//Verdichter zählen
	Count(
	x_Ein_1:= x_Aus1, 
	x_Ein_2:= x_Aus2, 
	x_Ein_3:= x_Aus3, 
	x_Ein_4:= x_Aus4,
	x_Ein_5:= x_Aus5,
	x_Ein_6:= x_Aus6,
	x_Ein_7:= x_Aus7,
	x_Ein_8:= x_Aus8,
	i_Aus=> i_Count);
//Betriebsstunden vergleichen
	//Vergleich zu Verdichter 1
	x_1_2(t_Ein1:=t_Betriebsstunden1, t_Ein2:= t_Betriebsstunden2);
	x_1_3(t_Ein1:=t_Betriebsstunden1, t_Ein2:= t_Betriebsstunden3);
	x_1_4(t_Ein1:=t_Betriebsstunden1, t_Ein2:= t_Betriebsstunden4);
	x_1_5(t_Ein1:=t_Betriebsstunden1, t_Ein2:= t_Betriebsstunden5);
	x_1_6(t_Ein1:=t_Betriebsstunden1, t_Ein2:= t_Betriebsstunden6);
	x_1_7(t_Ein1:=t_Betriebsstunden1, t_Ein2:= t_Betriebsstunden7);
	x_1_8(t_Ein1:=t_Betriebsstunden1, t_Ein2:= t_Betriebsstunden8);
	//Vergleich zu Verdichter 2
	x_2_1(t_Ein1:=t_Betriebsstunden2, t_Ein2:= t_Betriebsstunden1);
	x_2_3(t_Ein1:=t_Betriebsstunden2, t_Ein2:= t_Betriebsstunden3);
	x_2_4(t_Ein1:=t_Betriebsstunden2, t_Ein2:= t_Betriebsstunden4);
	x_2_5(t_Ein1:=t_Betriebsstunden2, t_Ein2:= t_Betriebsstunden5);
	x_2_6(t_Ein1:=t_Betriebsstunden2, t_Ein2:= t_Betriebsstunden6);
	x_2_7(t_Ein1:=t_Betriebsstunden2, t_Ein2:= t_Betriebsstunden7);
	x_2_8(t_Ein1:=t_Betriebsstunden2, t_Ein2:= t_Betriebsstunden8);
	//Vergleich zu Verdichter 3
	x_3_1(t_Ein1:=t_Betriebsstunden3, t_Ein2:= t_Betriebsstunden1);
	x_3_2(t_Ein1:=t_Betriebsstunden3, t_Ein2:= t_Betriebsstunden2);
	x_3_4(t_Ein1:=t_Betriebsstunden3, t_Ein2:= t_Betriebsstunden4);
	x_3_5(t_Ein1:=t_Betriebsstunden3, t_Ein2:= t_Betriebsstunden5);
	x_3_6(t_Ein1:=t_Betriebsstunden3, t_Ein2:= t_Betriebsstunden6);
	x_3_7(t_Ein1:=t_Betriebsstunden3, t_Ein2:= t_Betriebsstunden7);
	x_3_8(t_Ein1:=t_Betriebsstunden3, t_Ein2:= t_Betriebsstunden8);
	//Vergleich zu Verdichter 4
	x_4_1(t_Ein1:=t_Betriebsstunden4, t_Ein2:= t_Betriebsstunden1);
	x_4_2(t_Ein1:=t_Betriebsstunden4, t_Ein2:= t_Betriebsstunden2);
	x_4_3(t_Ein1:=t_Betriebsstunden4, t_Ein2:= t_Betriebsstunden3);
	x_4_5(t_Ein1:=t_Betriebsstunden4, t_Ein2:= t_Betriebsstunden5);
	x_4_6(t_Ein1:=t_Betriebsstunden4, t_Ein2:= t_Betriebsstunden6);
	x_4_7(t_Ein1:=t_Betriebsstunden4, t_Ein2:= t_Betriebsstunden7);
	x_4_8(t_Ein1:=t_Betriebsstunden4, t_Ein2:= t_Betriebsstunden8);
	//Vergleich zu Verdichter 5
	x_5_1(t_Ein1:=t_Betriebsstunden5, t_Ein2:= t_Betriebsstunden1);
	x_5_2(t_Ein1:=t_Betriebsstunden5, t_Ein2:= t_Betriebsstunden2);
	x_5_3(t_Ein1:=t_Betriebsstunden5, t_Ein2:= t_Betriebsstunden3);
	x_5_4(t_Ein1:=t_Betriebsstunden5, t_Ein2:= t_Betriebsstunden4);
	x_5_6(t_Ein1:=t_Betriebsstunden5, t_Ein2:= t_Betriebsstunden6);
	x_5_7(t_Ein1:=t_Betriebsstunden5, t_Ein2:= t_Betriebsstunden7);
	x_5_8(t_Ein1:=t_Betriebsstunden5, t_Ein2:= t_Betriebsstunden8);
	//Vergleich zu Verdichter 6
	x_6_1(t_Ein1:=t_Betriebsstunden6, t_Ein2:= t_Betriebsstunden1);
	x_6_2(t_Ein1:=t_Betriebsstunden6, t_Ein2:= t_Betriebsstunden2);
	x_6_3(t_Ein1:=t_Betriebsstunden6, t_Ein2:= t_Betriebsstunden3);
	x_6_4(t_Ein1:=t_Betriebsstunden6, t_Ein2:= t_Betriebsstunden4);
	x_6_5(t_Ein1:=t_Betriebsstunden6, t_Ein2:= t_Betriebsstunden5);
	x_6_7(t_Ein1:=t_Betriebsstunden6, t_Ein2:= t_Betriebsstunden7);
	x_6_8(t_Ein1:=t_Betriebsstunden6, t_Ein2:= t_Betriebsstunden8);
	//Vergleich zu Verdichter 7
	x_7_1(t_Ein1:=t_Betriebsstunden7, t_Ein2:= t_Betriebsstunden1);
	x_7_2(t_Ein1:=t_Betriebsstunden7, t_Ein2:= t_Betriebsstunden2);
	x_7_3(t_Ein1:=t_Betriebsstunden7, t_Ein2:= t_Betriebsstunden3);
	x_7_4(t_Ein1:=t_Betriebsstunden7, t_Ein2:= t_Betriebsstunden4);
	x_7_5(t_Ein1:=t_Betriebsstunden7, t_Ein2:= t_Betriebsstunden5);
	x_7_6(t_Ein1:=t_Betriebsstunden7, t_Ein2:= t_Betriebsstunden6);
	x_7_8(t_Ein1:=t_Betriebsstunden7, t_Ein2:= t_Betriebsstunden8);
	//Vergleich zu Verdichter 8
	x_8_1(t_Ein1:=t_Betriebsstunden8, t_Ein2:= t_Betriebsstunden1);
	x_8_2(t_Ein1:=t_Betriebsstunden8, t_Ein2:= t_Betriebsstunden2);
	x_8_3(t_Ein1:=t_Betriebsstunden8, t_Ein2:= t_Betriebsstunden3);
	x_8_4(t_Ein1:=t_Betriebsstunden8, t_Ein2:= t_Betriebsstunden4);
	x_8_5(t_Ein1:=t_Betriebsstunden8, t_Ein2:= t_Betriebsstunden5);
	x_8_6(t_Ein1:=t_Betriebsstunden8, t_Ein2:= t_Betriebsstunden6);
	x_8_7(t_Ein1:=t_Betriebsstunden8, t_Ein2:= t_Betriebsstunden7);
	
//Verdichterumschaltung für einen Zyklus einen Verdichter mehr anfordern Umschaltung verläuft also quasi nahtlos
	IF x_Wechsel AND NOT x_Speicher THEN
		i_Stufen:= i_Stufen+1;
	END_IF
	x_Speicher:=x_Wechsel;
	
//Einschalten
	//Einschalten Verdichter 1
		IF x_En1 AND i_Stufen > i_Count AND NOT x_Aus1 AND
			(x_1_2.x_Aus AND x_En2 OR x_Aus2 OR NOT x_En2) AND
			(x_1_3.x_Aus AND x_En3 OR x_Aus3 OR NOT x_En3) AND
			(x_1_4.x_Aus AND x_En4 OR x_Aus4 OR NOT x_En4) AND
			(x_1_5.x_Aus AND x_En5 OR x_Aus5 OR NOT x_En5) AND
			(x_1_6.x_Aus AND x_En6 OR x_Aus6 OR NOT x_En6) AND
			(x_1_7.x_Aus AND x_En7 OR x_Aus7 OR NOT x_En7) AND
			(x_1_8.x_Aus AND x_En8 OR x_Aus8 OR NOT x_En8) THEN
			x_Aus1:=TRUE;
			t_Ein1:=Globale_Uhr.systemDateAndTime;
			i_Count:=i_Count+1;
		END_IF
	
	//Einschalten Verdichter 2
		IF x_En2 AND i_Stufen > i_Count AND NOT x_Aus2 AND
			(x_2_1.x_Aus AND x_En1 OR x_Aus1 OR NOT x_En1) AND
			(x_2_3.x_Aus AND x_En3 OR x_Aus3 OR NOT x_En3) AND
			(x_2_4.x_Aus AND x_En4 OR x_Aus4 OR NOT x_En4) AND
			(x_2_5.x_Aus AND x_En5 OR x_Aus5 OR NOT x_En5) AND
			(x_2_6.x_Aus AND x_En6 OR x_Aus6 OR NOT x_En6) AND
			(x_2_7.x_Aus AND x_En7 OR x_Aus7 OR NOT x_En7) AND
			(x_2_8.x_Aus AND x_En8 OR x_Aus8 OR NOT x_En8) THEN
			x_Aus2:=TRUE;
			t_Ein2:=Globale_Uhr.systemDateAndTime;
			i_Count:=i_Count+1;
		END_IF	
	
	//Einschalten Verdichter 3
		IF x_En3 AND i_Stufen > i_Count AND NOT x_Aus3 AND
			(x_3_1.x_Aus AND x_En1 OR x_Aus1 OR NOT x_En1) AND
			(x_3_2.x_Aus AND x_En2 OR x_Aus2 OR NOT x_En2) AND
			(x_3_4.x_Aus AND x_En4 OR x_Aus4 OR NOT x_En4) AND
			(x_3_5.x_Aus AND x_En5 OR x_Aus5 OR NOT x_En5) AND
			(x_3_6.x_Aus AND x_En6 OR x_Aus6 OR NOT x_En6) AND
			(x_3_7.x_Aus AND x_En7 OR x_Aus7 OR NOT x_En7) AND
			(x_3_8.x_Aus AND x_En8 OR x_Aus8 OR NOT x_En8) THEN
			x_Aus3:=TRUE;
			t_Ein3:=Globale_Uhr.systemDateAndTime;
			i_Count:=i_Count+1;
		END_IF	
	
	//Einschalten Verdichter 4
		IF x_En4 AND i_Stufen > i_Count AND NOT x_Aus4 AND 
			(x_4_1.x_Aus AND x_En1 OR x_Aus1 OR NOT x_En1) AND
			(x_4_2.x_Aus AND x_En2 OR x_Aus2 OR NOT x_En2) AND
			(x_4_3.x_Aus AND x_En3 OR x_Aus3 OR NOT x_En3) AND
			(x_4_5.x_Aus AND x_En5 OR x_Aus5 OR NOT x_En5) AND
			(x_4_6.x_Aus AND x_En6 OR x_Aus6 OR NOT x_En6) AND
			(x_4_7.x_Aus AND x_En7 OR x_Aus7 OR NOT x_En7) AND
			(x_4_8.x_Aus AND x_En8 OR x_Aus8 OR NOT x_En8) THEN
			x_Aus4:=TRUE;
			t_Ein4:=Globale_Uhr.systemDateAndTime;
			i_Count:=i_Count+1;
		END_IF	
	//Einschalten Verdichter 5
		IF x_En5 AND i_Stufen > i_Count AND NOT x_Aus5 AND
			(x_5_1.x_Aus AND x_En1 OR x_Aus1 OR NOT x_En1) AND
			(x_5_2.x_Aus AND x_En2 OR x_Aus2 OR NOT x_En2) AND
			(x_5_3.x_Aus AND x_En3 OR x_Aus3 OR NOT x_En3) AND
			(x_5_4.x_Aus AND x_En4 OR x_Aus4 OR NOT x_En4) AND
			(x_5_6.x_Aus AND x_En6 OR x_Aus6 OR NOT x_En6) AND
			(x_5_7.x_Aus AND x_En7 OR x_Aus7 OR NOT x_En7) AND
			(x_5_8.x_Aus AND x_En8 OR x_Aus8 OR NOT x_En8) THEN
			x_Aus5:=TRUE;
			t_Ein5:=Globale_Uhr.systemDateAndTime;
			i_Count:=i_Count+1;
		END_IF
	
	//Einschalten Verdichter 6
		IF x_En6 AND i_Stufen > i_Count AND NOT x_Aus6 AND
			(x_6_1.x_Aus AND x_En1 OR x_Aus1 OR NOT x_En1) AND
			(x_6_2.x_Aus AND x_En2 OR x_Aus2 OR NOT x_En2) AND
			(x_6_3.x_Aus AND x_En3 OR x_Aus3 OR NOT x_En3) AND
			(x_6_4.x_Aus AND x_En4 OR x_Aus4 OR NOT x_En4) AND
			(x_6_5.x_Aus AND x_En5 OR x_Aus5 OR NOT x_En5) AND
			(x_6_7.x_Aus AND x_En7 OR x_Aus7 OR NOT x_En7) AND
			(x_6_8.x_Aus AND x_En8 OR x_Aus8 OR NOT x_En8) THEN
			x_Aus6:=TRUE;
			t_Ein6:=Globale_Uhr.systemDateAndTime;
			i_Count:=i_Count+1;
		END_IF	
	
	//Einschalten Verdichter 7
		IF x_En7 AND i_Stufen > i_Count AND NOT x_Aus7 AND
			(x_7_1.x_Aus AND x_En1 OR x_Aus1 OR NOT x_En1) AND
			(x_7_2.x_Aus AND x_En2 OR x_Aus2 OR NOT x_En2) AND
			(x_7_3.x_Aus AND x_En3 OR x_Aus3 OR NOT x_En3) AND
			(x_7_4.x_Aus AND x_En4 OR x_Aus4 OR NOT x_En4) AND
			(x_7_5.x_Aus AND x_En5 OR x_Aus5 OR NOT x_En5) AND
			(x_7_6.x_Aus AND x_En6 OR x_Aus6 OR NOT x_En6) AND
			(x_7_8.x_Aus AND x_En8 OR x_Aus8 OR NOT x_En8) THEN
			x_Aus7:=TRUE;
			t_Ein7:=Globale_Uhr.systemDateAndTime;
			i_Count:=i_Count+1;
		END_IF	
	
	//Einschalten Verdichter 8
		IF x_En8 AND i_Stufen > i_Count AND NOT x_Aus8 AND
			(x_8_1.x_Aus AND x_En1 OR x_Aus1 OR NOT x_En1) AND
			(x_8_2.x_Aus AND x_En2 OR x_Aus2 OR NOT x_En2) AND
			(x_8_3.x_Aus AND x_En3 OR x_Aus3 OR NOT x_En3) AND
			(x_8_4.x_Aus AND x_En4 OR x_Aus4 OR NOT x_En4) AND
			(x_8_5.x_Aus AND x_En5 OR x_Aus5 OR NOT x_En5) AND
			(x_8_6.x_Aus AND x_En6 OR x_Aus6 OR NOT x_En6) AND
			(x_8_7.x_Aus AND x_En7 OR x_Aus7 OR NOT x_En7) THEN
			x_Aus8:=TRUE;
			t_Ein8:=Globale_Uhr.systemDateAndTime;
			i_Count:=i_Count+1;
		END_IF	
	
//Ausschalten
	//Ausschalten Verdichter 1
		IF NOT x_En1 AND x_Aus1 OR (i_Stufen < i_Count AND x_Aus1 AND
			//(t_Ein1 <= t_Ein1 OR NOT x_Aus1) AND
			(t_Ein1 <= t_Ein2 OR NOT x_Aus2) AND
			(t_Ein1 <= t_Ein3 OR NOT x_Aus3) AND
			(t_Ein1 <= t_Ein4 OR NOT x_Aus4) AND
			(t_Ein1 <= t_Ein5 OR NOT x_Aus5) AND
			(t_Ein1 <= t_Ein6 OR NOT x_Aus6) AND
			(t_Ein1 <= t_Ein7 OR NOT x_Aus7) AND
			(t_Ein1 <= t_Ein8 OR NOT x_Aus8)) THEN
			x_Aus1:=FALSE;
			i_Count:= i_Count-1;
		END_IF	
		
	//Ausschalten Verdichter 2
		IF NOT x_En2 AND x_Aus2 OR (i_Stufen < i_Count AND x_Aus2 AND
			(t_Ein2 <= t_Ein1 OR NOT x_Aus1) AND
			//(t_Ein2 <= t_Ein2 OR NOT x_Aus2) AND
			(t_Ein2 <= t_Ein3 OR NOT x_Aus3) AND
			(t_Ein2 <= t_Ein4 OR NOT x_Aus4) AND
			(t_Ein2 <= t_Ein5 OR NOT x_Aus5) AND
			(t_Ein2 <= t_Ein6 OR NOT x_Aus6) AND
			(t_Ein2 <= t_Ein7 OR NOT x_Aus7) AND
			(t_Ein2 <= t_Ein8 OR NOT x_Aus8)) THEN
			x_Aus2:=FALSE;
			i_Count:= i_Count-1;
		END_IF	
		
	//Ausschalten Verdichter 3
		IF NOT x_En3 AND x_Aus3 OR (i_Stufen < i_Count AND x_Aus3 AND
			(t_Ein3 <= t_Ein1 OR NOT x_Aus1) AND
			(t_Ein3 <= t_Ein2 OR NOT x_Aus2) AND
			//(t_Ein3 <= t_Ein3 OR NOT x_Aus3) AND
			(t_Ein3 <= t_Ein4 OR NOT x_Aus4) AND
			(t_Ein3 <= t_Ein5 OR NOT x_Aus5) AND
			(t_Ein3 <= t_Ein6 OR NOT x_Aus6) AND
			(t_Ein3 <= t_Ein7 OR NOT x_Aus7) AND
			(t_Ein3 <= t_Ein8 OR NOT x_Aus8)) THEN
			x_Aus3:=FALSE;
			i_Count:= i_Count-1;
		END_IF	
		
	//Ausschalten Verdichter 4
		IF NOT x_En4 AND x_Aus4 OR (i_Stufen < i_Count AND x_Aus4 AND
			(t_Ein4 <= t_Ein1 OR NOT x_Aus1) AND
			(t_Ein4 <= t_Ein2 OR NOT x_Aus2) AND
			(t_Ein4 <= t_Ein3 OR NOT x_Aus3) AND
			//(t_Ein4 <= t_Ein4 OR NOT x_Aus4) AND
			(t_Ein4 <= t_Ein5 OR NOT x_Aus5) AND
			(t_Ein4 <= t_Ein6 OR NOT x_Aus6) AND
			(t_Ein4 <= t_Ein7 OR NOT x_Aus7) AND
			(t_Ein4 <= t_Ein8 OR NOT x_Aus8)) THEN
			x_Aus4:=FALSE;
			i_Count:= i_Count-1;
		END_IF	
		
	//Ausschalten Verdichter 5
		IF NOT x_En5 AND x_Aus5 OR (i_Stufen < i_Count AND x_Aus5 AND
			(t_Ein5 <= t_Ein1 OR NOT x_Aus1) AND
			(t_Ein5 <= t_Ein2 OR NOT x_Aus2) AND
			(t_Ein5 <= t_Ein3 OR NOT x_Aus3) AND
			(t_Ein5 <= t_Ein4 OR NOT x_Aus4) AND
			//(t_Ein5 <= t_Ein5 OR NOT x_Aus5) AND
			(t_Ein5 <= t_Ein6 OR NOT x_Aus6) AND
			(t_Ein5 <= t_Ein7 OR NOT x_Aus7) AND
			(t_Ein5 <= t_Ein8 OR NOT x_Aus8)) THEN
			x_Aus5:=FALSE;
			i_Count:= i_Count-1;
		END_IF		
		
	//Ausschalten Verdichter 6
		IF NOT x_En6 AND x_Aus6 OR (i_Stufen < i_Count AND x_Aus6 AND
			(t_Ein6 <= t_Ein1 OR NOT x_Aus1) AND
			(t_Ein6 <= t_Ein2 OR NOT x_Aus2) AND
			(t_Ein6 <= t_Ein3 OR NOT x_Aus3) AND
			(t_Ein6 <= t_Ein4 OR NOT x_Aus4) AND
			(t_Ein6 <= t_Ein5 OR NOT x_Aus5) AND
			//(t_Ein6 <= t_Ein6 OR NOT x_Aus6) AND
			(t_Ein6 <= t_Ein7 OR NOT x_Aus7) AND
			(t_Ein6 <= t_Ein8 OR NOT x_Aus8)) THEN
			x_Aus6:=FALSE;
			i_Count:= i_Count-1;
		END_IF	
		
	//Ausschalten Verdichter 7
		IF NOT x_En7 AND x_Aus7 OR (i_Stufen < i_Count AND x_Aus7 AND
			(t_Ein7 <= t_Ein1 OR NOT x_Aus1) AND
			(t_Ein7 <= t_Ein2 OR NOT x_Aus2) AND
			(t_Ein7 <= t_Ein3 OR NOT x_Aus3) AND
			(t_Ein7 <= t_Ein4 OR NOT x_Aus4) AND
			(t_Ein7 <= t_Ein5 OR NOT x_Aus5) AND
			(t_Ein7 <= t_Ein6 OR NOT x_Aus6) AND
			//(t_Ein7 <= t_Ein7 OR NOT x_Aus7) AND
			(t_Ein7 <= t_Ein8 OR NOT x_Aus8)) THEN
			x_Aus7:=FALSE;
			i_Count:= i_Count-1;
		END_IF	
		
	//Ausschalten Verdichter 8
		IF NOT x_En8 AND x_Aus8 OR (i_Stufen < i_Count AND x_Aus8 AND
			(t_Ein8 <= t_Ein1 OR NOT x_Aus1) AND
			(t_Ein8 <= t_Ein2 OR NOT x_Aus2) AND
			(t_Ein8 <= t_Ein3 OR NOT x_Aus3) AND
			(t_Ein8 <= t_Ein4 OR NOT x_Aus4) AND
			(t_Ein8 <= t_Ein5 OR NOT x_Aus5) AND
			(t_Ein8 <= t_Ein6 OR NOT x_Aus6) AND
			(t_Ein8 <= t_Ein7 OR NOT x_Aus7) (*AND
			(t_Ein8 <= t_Ein8 OR NOT x_Aus8) *))THEN
			x_Aus8:=FALSE;
			i_Count:= i_Count-1;
		END_IF

END_FUNCTION_BLOCK

// Verdichter/Verdichter
FUNCTION_BLOCK Verdichter
VAR_INPUT
END_VAR
VAR_OUTPUT
END_VAR
VAR
	x_Steuerschalter: BOOL;
	x_Betrieb: BOOL;
	x_Stoerung: BOOL;
	t_Betriebsstunden:timestruct;
	i_Einschaltungen: INT;
	t_RestZeitWiedereinschaltsperre:timestruct;
	x_ResetWiedereinschaltsperre: BOOL;
	t_Wiedereinschaltsperre:timestruct;
	t_StartBetriebsstunden:Timestruct;//Betriebsstunden die beim Reset geschrieben werden
	i_StartEinschaltungen:INT;//Impulse die beim Reset geschrieben werden
	f_MinOeldruckDifferenz: REAL;
	t_AlarmOeldruck:timestruct;
END_VAR

// NETWORK 1

END_FUNCTION_BLOCK

// Verdichter/SA_Scroll
(*Funktionsbaustein für einen Scrollverdichter mit Sanftanlauf. 
*)
FUNCTION_BLOCK SA_Scroll
(*
Versionsverlauf: 
Version		|Autor	|Bemerkung
------------------------------------------------------------------------------------------------------------ 
17.06.00	|Shgb	|erste Freigabe 
17.08.00	|LeaF	|Freigabe

*)
VAR_INPUT 
	x_HD_Pressostat :BOOL;//Rückmeldung des Hochdruckpressostates
	x_RM_Sanftanlauf:BOOL;//Rückmeldung vom Sanfanlauf als Betriebsmeldung
	x_Einschaltbefehl:BOOL;//Einschaltbefehl für den Kompressor
	x_Quittieren:BOOL;//Quittieren der Alarme
	x_ResetWiedereinschaltsperre:BOOL;//Wiedereinschaltsprerre quittieren
	x_ResetBetriebsstunden:BOOL;//Betriebsstunden zurücksetzen
	x_FG_Ext:BOOL:=TRUE;//Externe Freigabe
END_VAR
VAR_INPUT PERSISTENT
	x_SoftSchalter:BOOL;//Handschaltung für Visu
	t_Wiedereinschaltsperre:timestruct := (wMinute := 15);	//Sollzeit für die Wiedereinschaltsperre
	t_StartBetriebsstunden:Timestruct;//Betriebsstunden die beim Reset geschrieben werden
	i_StartEinschaltungen:INT;//Impulse die beim Reset geschrieben werden
END_VAR
VAR_OUTPUT
	x_Freigabe:BOOL;//Kompressor ist Freigegeben
	t_RestzeitWiedereinschaltsperre:timestruct;//Restzeit der Wiedereinschaltsperre
	t_Betriebsstunden:timestruct;//Betriebsstunden des Kompressors
	i_Einschaltungen:INT;//Einschaltimpulse des Kompressors
	x_Kompressor:BOOL;//Einschaltbefehl für den Kompressor
	x_AL_Sanftanlauf:BOOL;//Alarm keine Betriebsmeldung durch Sanftanlauf
	x_AL_HD_Pressostat:BOOL;//Alarm keine Rückmeldung durch Hochdruckpressostat
END_VAR
VAR
	x_Wiedereinschaltsperre,x_Alarme,x_Temp: BOOL;
	Wiedereinschaltsperre: TOF_Reset;
	TON_Sanftanlauf: TON;
	Work: Work;
	x_Speicher: BOOL;
END_VAR

//Alarme
	//Alle Alarme müssen vor dem zyklischen Ablauf geprüft werden.
	//Quittieren
	IF x_Quittieren THEN
		x_AL_HD_Pressostat:=FALSE;
		x_AL_Sanftanlauf:=FALSE;
	END_IF
	
	//Hochdruckpressostat
	IF NOT x_HD_Pressostat THEN
		x_AL_HD_Pressostat:= TRUE;
	END_IF
	
	//Rückmeldung Sanftanlauf
	TON_Sanftanlauf(IN:=x_Kompressor AND NOT x_RM_Sanftanlauf, PT:= T#1S, Q=> x_Temp, ET=> );
	IF x_Temp THEN
		x_AL_Sanftanlauf:= TRUE;	
	END_IF
	
	x_Alarme:=x_AL_Sanftanlauf OR x_AL_HD_Pressostat;
	
//Verdichterfreigabe 
	x_Freigabe := x_SoftSchalter AND x_FG_Ext AND NOT x_Wiedereinschaltsperre AND NOT x_Alarme;
	
//Wiedereinschaltsperre
	Wiedereinschaltsperre(
		x_Ein:= NOT x_Kompressor AND x_Speicher, 
		x_Reset:= x_ResetWiedereinschaltsperre, 
		t_time:= t_Wiedereinschaltsperre, 
		x_Aus=> x_Wiedereinschaltsperre, 
		t_Restzeit=> t_RestzeitWiedereinschaltsperre);
	x_Speicher:=x_Kompressor;
		
//Einschaltbefehl
	x_Kompressor:= x_Einschaltbefehl AND x_Freigabe;
	
//Betriebsstunden
	Work(x_Ein:= x_Kompressor,
		x_Reset:= x_ResetBetriebsstunden,
		t_StartBetriebsstunden:=t_StartBetriebsstunden,
		i_StartEinschaltungen:=i_StartEinschaltungen,
		t_Betriebsstunden=> t_Betriebsstunden, 
		i_Einschaltungen=> i_Einschaltungen);

END_FUNCTION_BLOCK

(* text list Alarme (id | default | Deutsch)
  0 | ID0 | 
  1 | ID1 | 
  2 | ID2 | 
  3 | ID3 | 
  4 | ID4 | 
  5 | ID5 | 
  6 | ID6 | 
  7 | ID7 | 
  8 | ID8 | 
  9 | ID9 | 
  10 | ID10 | 
  11 | ID11 | 
  12 | ID12 | 
  13 | ID13 | 
  14 | ID14 | 
  15 | ID15 | 
  16 | ID16 | 
  17 | ID17 | 
  18 | ID18 | 
  19 | ID19 | 
  20 | ID20 | 
  21 | ID21 | 
  22 | ID22 | 
  23 | ID23 | 
  24 | ID24 | 
  25 | ID25 | 
  26 | ID26 | 
  27 | ID27 | 
  28 | ID28 | 
  29 | ID29 | 
  30 | ID30 | 
  31 | ID31 | 
  32 | ID32 | 
  33 | ID33 | 
  34 | ID34 | 
  35 | ID35 | 
  36 | ID36 | 
  37 | ID37 | 
  38 | ID38 | 
  39 | ID39 | 
  40 | ID40 | 
  41 | ID41 | 
  42 | ID42 | 
  43 | ID43 | 
  44 | ID44 | 
  45 | ID45 | 
  46 | ID46 | 
  47 | ID47 | 
  48 | ID48 | 
  49 | ID49 | 
  50 | ID50 | 
  51 | ID51 | 
  52 | ID52 | 
  53 | ID53 | 
  54 | ID54 | 
  55 | ID55 | 
  56 | ID56 | 
  57 | ID57 | 
  58 | ID58 | 
  59 | ID59 | 
  60 | ID60 | 
  61 | ID61 | 
  62 | ID62 | 
  63 | ID63 | 
  64 | ID64 | 
  65 | ID65 | 
  66 | ID66 | 
  67 | ID67 | 
  68 | ID68 | 
  69 | ID69 | 
  70 | ID70 | 
  71 | ID71 | 
  72 | ID72 | 
  73 | ID73 | 
  74 | ID74 | 
  75 | ID75 | 
  76 | ID76 | 
  77 | ID77 | 
  78 | ID78 | 
  79 | ID79 | 
  80 | ID80 | 
  81 | ID81 | 
  82 | ID82 | 
  83 | ID83 | 
  84 | ID84 | 
  85 | ID85 | 
  86 | ID86 | 
  87 | ID87 | 
  88 | ID88 | 
  89 | ID89 | 
  90 | ID90 | 
  91 | ID91 | 
  92 | ID92 | 
  93 | ID93 | 
  94 | ID94 | 
  95 | ID95 | 
  96 | ID96 | 
  97 | ID97 | 
  98 | ID98 | 
  99 | ID99 | 
   |  |  *)
